// SIMATIC S7-200 project (STEP 7-Micro/WIN), CPU 224 REL 02.01

SYMBOL_TABLE 用户定义1
I0_0             I0.0     // 输入信号
I0_1             I0.1     // 设备运行信号
M0_0             M0.0     // 输入信号上升延微分
M0_1             M0.1     // 输入信号下降延微分
M1_1             M1.1     // 输入信号有效上升延微分
M1_2             M1.2     // 输入信号有效下降延微分
M14_0            M14.0    // 输入信号状态保持
M14_1            M14.1    // 第1路输入信号保持状态1
M14_2            M14.2    // 第2路输入信号保持状态1
M14_3            M14.3    // 第3路输入信号保持状态1
M15_1            M15.1    // 第1路输入信号上升延微分
M15_2            M15.2    // 第2路输入信号上升延微分
M15_3            M15.3    // 第3路输入信号上升延微分
M16_1            M16.1    // 第1路输入信号保持状态2
M16_2            M16.2    // 第1路输入信号保持状态2
M16_3            M16.3    // 第3路输入信号保持状态2
M17_1            M17.1    // 延迟输出保持状态
Q0_0             Q0.0     // 延迟输出信号
T_10             T10      // 输入信号动作时间
T_11             T11      // 第1路输入信号动作时间
T_12             T12      // 第2路输入信号动作时间
T_13             T13      // 第3路输入信号动作时间
T_91             T91      // 再现输入动作时间
VW_10            VW10     // 第1路输入信号动作时间
VW_20            VW20     // 第2路输入信号动作时间
VW_30            VW30     // 第3路输入信号动作时间
VW_100           VW100    // 再现输入动作时间
END_SYMBOL_TABLE

ORGANIZATION_BLOCK 主程序:OB1
TITLE=该程序可以实现输入延迟一定时间后输出，而且延时输出时会再现输入动作时间；
// 该程序仅适合于输入信号持续时间比延迟输出时间短的情况，也适合于输入信号持续时间比延迟输出时间长的情况；
// 该程序因为采用了100ms定时器的原因，只有小于3276.7秒的持续输入会被响应，大于3276.7秒的持续输入将会被视作3276.7秒；
// 该程序具有断电保持功能。
// 该程序为记忆3个输入信号的示例程序：最多可以同时记忆3个输入信号，其余的输入信号将会被忽略；也就是说，如果延迟输出时间为X秒，那么在任意一个X秒的时间段范围以内，最多只能有3个输入信号有效（被记忆），其余的输入信号将会被忽略；
// 如果希望记忆N个输入信号，将程序进行相应扩展即可；
// 对于每个输入信号而言，其延迟输出时间都是一样的，否则就没有任何意义了（从逻辑上来说，根本无法对某个指定的输入信号分配延迟输出时间）；
// 该示例程序的延迟输出时间为10秒，控制精度为0.1S；如果希望控制精度更高、延迟输出时间更长，请采用相应的定时器；如果无法找到合适的定时器，请采用和控制精度级别相同的定时器+多个计数器级联来实现。
BEGIN
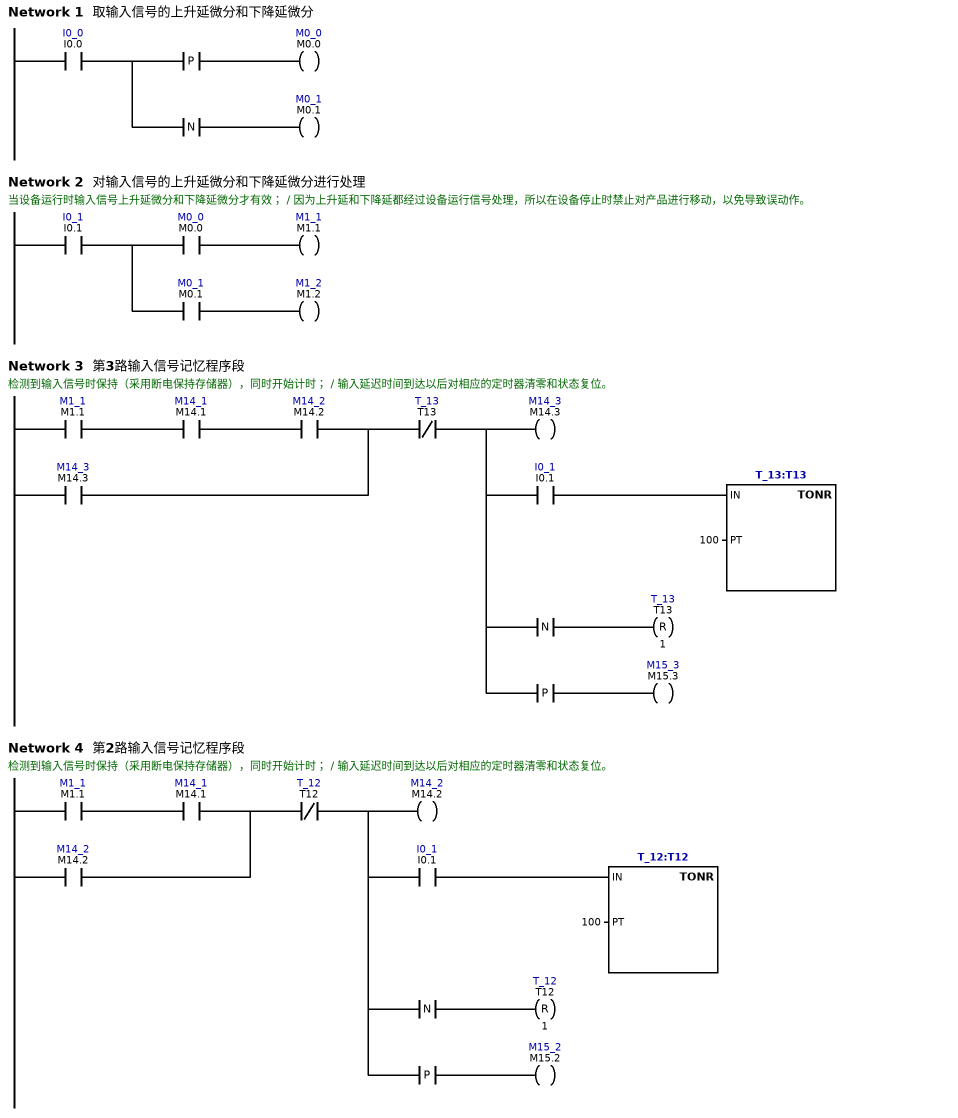
Network 1 // 取输入信号的上升延微分和下降延微分
LD     I0_0:I0.0
LPS
EU
=      M0_0:M0.0
LPP
ED
=      M0_1:M0.1
Network 2 // 对输入信号的上升延微分和下降延微分进行处理
// 当设备运行时输入信号上升延微分和下降延微分才有效；
// 因为上升延和下降延都经过设备运行信号处理，所以在设备停止时禁止对产品进行移动，以免导致误动作。
LD     I0_1:I0.1
LPS
A      M0_0:M0.0
=      M1_1:M1.1
LPP
A      M0_1:M0.1
=      M1_2:M1.2
Network 3 // 第3路输入信号记忆程序段
// 检测到输入信号时保持（采用断电保持存储器），同时开始计时；
// 输入延迟时间到达以后对相应的定时器清零和状态复位。
LD     M1_1:M1.1
A      M14_1:M14.1
A      M14_2:M14.2
O      M14_3:M14.3
AN     T_13:T13
LPS
=      M14_3:M14.3
A      I0_1:I0.1
TONR   T_13:T13, 100
LRD
ED
R      T_13:T13, 1
LPP
EU
=      M15_3:M15.3
Network 4 // 第2路输入信号记忆程序段
// 检测到输入信号时保持（采用断电保持存储器），同时开始计时；
// 输入延迟时间到达以后对相应的定时器清零和状态复位。
LD     M1_1:M1.1
A      M14_1:M14.1
O      M14_2:M14.2
AN     T_12:T12
LPS
=      M14_2:M14.2
A      I0_1:I0.1
TONR   T_12:T12, 100
LRD
ED
R      T_12:T12, 1
LPP
EU
=      M15_2:M15.2
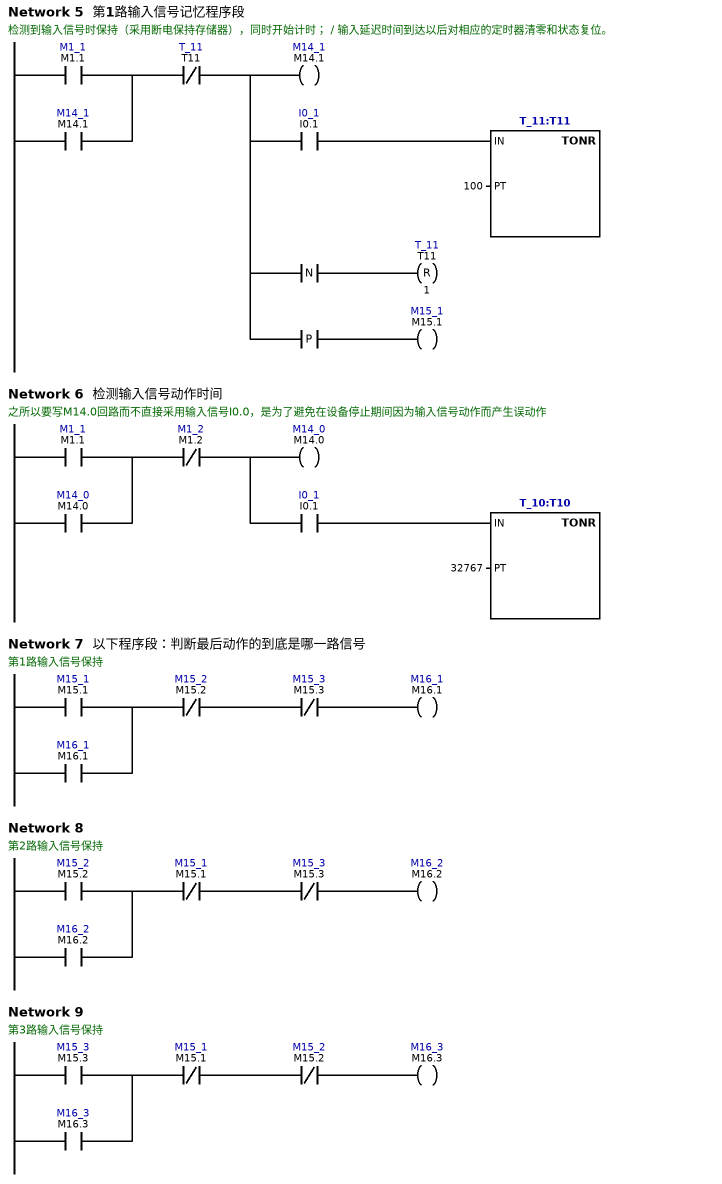
Network 5 // 第1路输入信号记忆程序段
// 检测到输入信号时保持（采用断电保持存储器），同时开始计时；
// 输入延迟时间到达以后对相应的定时器清零和状态复位。
LD     M1_1:M1.1
O      M14_1:M14.1
AN     T_11:T11
LPS
=      M14_1:M14.1
A      I0_1:I0.1
TONR   T_11:T11, 100
LRD
ED
R      T_11:T11, 1
LPP
EU
=      M15_1:M15.1
Network 6 // 检测输入信号动作时间
// 之所以要写M14.0回路而不直接采用输入信号I0.0，是为了避免在设备停止期间因为输入信号动作而产生误动作
LD     M1_1:M1.1
O      M14_0:M14.0
AN     M1_2:M1.2
=      M14_0:M14.0
A      I0_1:I0.1
TONR   T_10:T10, 32767
Network 7 // 以下程序段：判断最后动作的到底是哪一路信号
// 第1路输入信号保持
LD     M15_1:M15.1
O      M16_1:M16.1
AN     M15_2:M15.2
AN     M15_3:M15.3
=      M16_1:M16.1
Network 8
// 第2路输入信号保持
LD     M15_2:M15.2
O      M16_2:M16.2
AN     M15_1:M15.1
AN     M15_3:M15.3
=      M16_2:M16.2
Network 9
// 第3路输入信号保持
LD     M15_3:M15.3
O      M16_3:M16.3
AN     M15_1:M15.1
AN     M15_2:M15.2
=      M16_3:M16.3
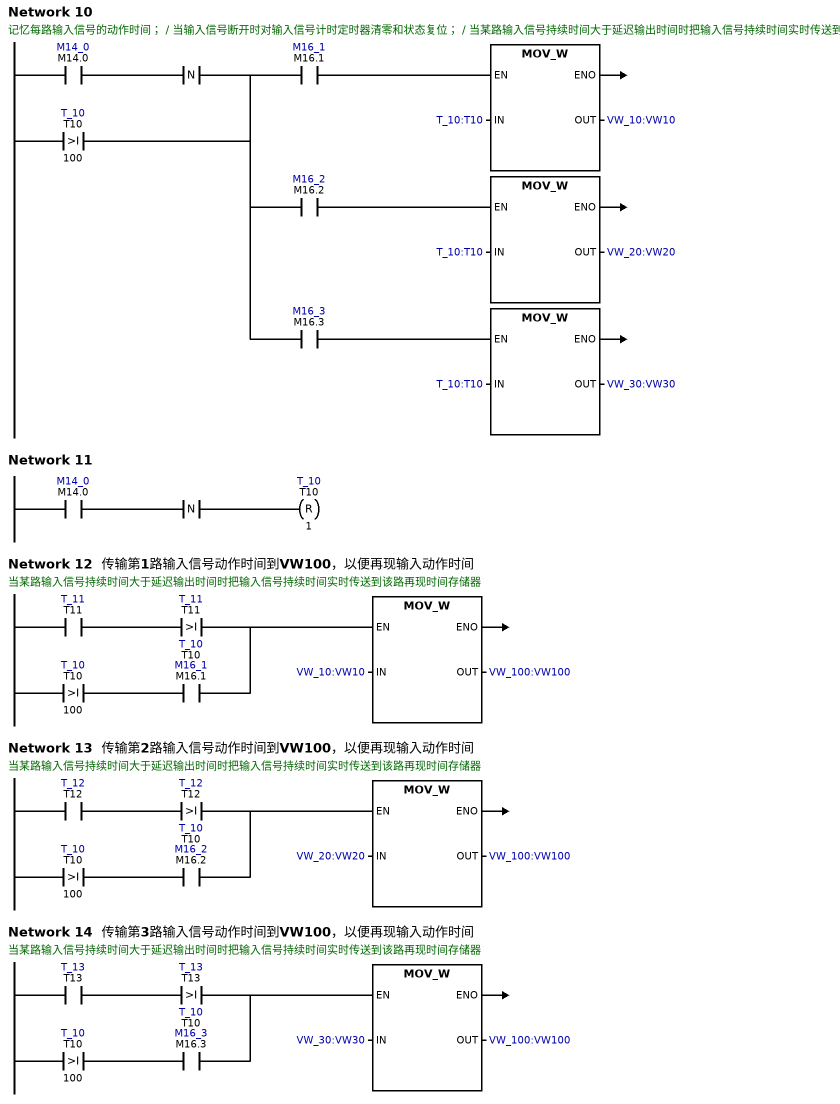
Network 10
// 记忆每路输入信号的动作时间；
// 当输入信号断开时对输入信号计时定时器清零和状态复位；
// 当某路输入信号持续时间大于延迟输出时间时把输入信号持续时间实时传送到该路再现时间存储器。
LD     M14_0:M14.0
ED
OW>    T_10:T10, 100
LPS
A      M16_1:M16.1
MOVW   T_10:T10, VW_10:VW10
LRD
A      M16_2:M16.2
MOVW   T_10:T10, VW_20:VW20
LPP
A      M16_3:M16.3
MOVW   T_10:T10, VW_30:VW30
Network 11
LD     M14_0:M14.0
ED
R      T_10:T10, 1
Network 12 // 传输第1路输入信号动作时间到VW100，以便再现输入动作时间
// 当某路输入信号持续时间大于延迟输出时间时把输入信号持续时间实时传送到该路再现时间存储器
LD     T_11:T11
AW>    T_11:T11, T_10:T10
LDW>   T_10:T10, 100
A      M16_1:M16.1
OLD
MOVW   VW_10:VW10, VW_100:VW100
Network 13 // 传输第2路输入信号动作时间到VW100，以便再现输入动作时间
// 当某路输入信号持续时间大于延迟输出时间时把输入信号持续时间实时传送到该路再现时间存储器
LD     T_12:T12
AW>    T_12:T12, T_10:T10
LDW>   T_10:T10, 100
A      M16_2:M16.2
OLD
MOVW   VW_20:VW20, VW_100:VW100
Network 14 // 传输第3路输入信号动作时间到VW100，以便再现输入动作时间
// 当某路输入信号持续时间大于延迟输出时间时把输入信号持续时间实时传送到该路再现时间存储器
LD     T_13:T13
AW>    T_13:T13, T_10:T10
LDW>   T_10:T10, 100
A      M16_3:M16.3
OLD
MOVW   VW_30:VW30, VW_100:VW100
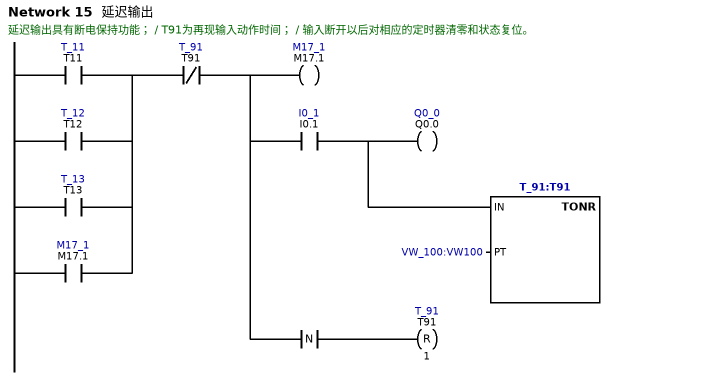
Network 15 // 延迟输出
// 延迟输出具有断电保持功能；
// T91为再现输入动作时间；
// 输入断开以后对相应的定时器清零和状态复位。
LD     T_11:T11
O      T_12:T12
O      T_13:T13
O      M17_1:M17.1
AN     T_91:T91
LPS
=      M17_1:M17.1
A      I0_1:I0.1
=      Q0_0:Q0.0
TONR   T_91:T91, VW_100:VW100
LPP
ED
R      T_91:T91, 1
END_ORGANIZATION_BLOCK
